{attribute 'qualified_only'}
VAR_GLOBAL	
	B1	 AT %I* :BOOL;   	// 	Füllstand Ölbehälter
	B2	 AT %I* :BOOL;   	// 	Öldruck erreicht
	B3	 AT %I* :BOOL;   	// 	Überdruck
	B4	 AT %I* :BOOL;   	// 	Temperatur Ölbehälter
	B5	 AT %I* :BOOL;   	// 	Druckschalter Ölfilter
	F1	 AT %I* :BOOL;   	// 	Thermorelais Motor
	S1	 AT %I* :BOOL;   	// 	Taster Start
	S2	 AT %I* :BOOL;   	// 	Taster Stop
	S3	 AT %I* :BOOL;   	// 	Taster Quittieren
	S4	 AT %I* :BOOL;   	// 	Taster Zylinder
END_VAR

(* stored: Version 1.1.0.1, ProductVersion 3.1.4024.5
   GVL DI: Id {c2d05302-d374-4f85-80dd-41006a3e3277} *)
